PROGRAM MAIN
VAR
END_VAR

RunMotor();

END_PROGRAM

(* stored: Version 1.1.0.1, ProductVersion 3.1.4024.12
   POU MAIN: Id {40408346-86d7-49f3-b513-34c5fb5b1363}, SpecialFunc None *)
